SUBAPPLICATION InputOutputTesterButton_PI_OPC_UA (* PI Tester (OPC-UA): 8 Puls-Eingaenge (Zaehler+Frequenz+Bargraph) + 12 unveraenderte digitale Ausgaenge *)
  (* Standard: 61499-2; Description: Copyright (c) 2026 Meisterschulen am Ostbahnhof This program and the accompanying materials are made available under the terms of the Eclipse Public License 2.0 which is available at https://www.eclipse.org/legal/epl-2.0/ SPDX-License-Identifier: EPL-2.0 *)
  (* Version 1.0, 2026-08-30, Franz Höpfinger, Meisterschulen am Ostbahnhof, initial API and implementation and/or initial documentation *)
  PACKAGE Meins::InputOutputTester::Button_PI_OPC_UA;
  IMPORT Meins::InputOutputTester::Button_PI_OPC_UA::SubStrings::PI_I1_COUNT_WRITE;
  IMPORT Meins::InputOutputTester::Button_PI_OPC_UA::SubStrings::PI_I1_FREQ_WRITE;
  IMPORT Meins::InputOutputTester::Button_PI_OPC_UA::SubStrings::PI_I1_SWITCH_READ;
  IMPORT Meins::InputOutputTester::Button_PI_OPC_UA::SubStrings::PI_I1_SWITCH_WRITE;
  IMPORT Meins::InputOutputTester::Button_PI_OPC_UA::SubStrings::PI_I1_STATUS_WRITE;
  IMPORT Meins::InputOutputTester::Button_PI_OPC_UA::SubStrings::PI_I2_COUNT_WRITE;
  IMPORT Meins::InputOutputTester::Button_PI_OPC_UA::SubStrings::PI_I2_FREQ_WRITE;
  IMPORT Meins::InputOutputTester::Button_PI_OPC_UA::SubStrings::PI_I2_SWITCH_READ;
  IMPORT Meins::InputOutputTester::Button_PI_OPC_UA::SubStrings::PI_I2_SWITCH_WRITE;
  IMPORT Meins::InputOutputTester::Button_PI_OPC_UA::SubStrings::PI_I2_STATUS_WRITE;
  IMPORT Meins::InputOutputTester::Button_PI_OPC_UA::SubStrings::PI_I3_COUNT_WRITE;
  IMPORT Meins::InputOutputTester::Button_PI_OPC_UA::SubStrings::PI_I3_FREQ_WRITE;
  IMPORT Meins::InputOutputTester::Button_PI_OPC_UA::SubStrings::PI_I3_SWITCH_READ;
  IMPORT Meins::InputOutputTester::Button_PI_OPC_UA::SubStrings::PI_I3_SWITCH_WRITE;
  IMPORT Meins::InputOutputTester::Button_PI_OPC_UA::SubStrings::PI_I3_STATUS_WRITE;
  IMPORT Meins::InputOutputTester::Button_PI_OPC_UA::SubStrings::PI_I4_COUNT_WRITE;
  IMPORT Meins::InputOutputTester::Button_PI_OPC_UA::SubStrings::PI_I4_FREQ_WRITE;
  IMPORT Meins::InputOutputTester::Button_PI_OPC_UA::SubStrings::PI_I4_SWITCH_READ;
  IMPORT Meins::InputOutputTester::Button_PI_OPC_UA::SubStrings::PI_I4_SWITCH_WRITE;
  IMPORT Meins::InputOutputTester::Button_PI_OPC_UA::SubStrings::PI_I4_STATUS_WRITE;
  IMPORT Meins::InputOutputTester::Button_PI_OPC_UA::SubStrings::PI_I5_COUNT_WRITE;
  IMPORT Meins::InputOutputTester::Button_PI_OPC_UA::SubStrings::PI_I5_FREQ_WRITE;
  IMPORT Meins::InputOutputTester::Button_PI_OPC_UA::SubStrings::PI_I5_SWITCH_READ;
  IMPORT Meins::InputOutputTester::Button_PI_OPC_UA::SubStrings::PI_I5_SWITCH_WRITE;
  IMPORT Meins::InputOutputTester::Button_PI_OPC_UA::SubStrings::PI_I5_STATUS_WRITE;
  IMPORT Meins::InputOutputTester::Button_PI_OPC_UA::SubStrings::PI_I6_COUNT_WRITE;
  IMPORT Meins::InputOutputTester::Button_PI_OPC_UA::SubStrings::PI_I6_FREQ_WRITE;
  IMPORT Meins::InputOutputTester::Button_PI_OPC_UA::SubStrings::PI_I6_SWITCH_READ;
  IMPORT Meins::InputOutputTester::Button_PI_OPC_UA::SubStrings::PI_I6_SWITCH_WRITE;
  IMPORT Meins::InputOutputTester::Button_PI_OPC_UA::SubStrings::PI_I6_STATUS_WRITE;
  IMPORT Meins::InputOutputTester::Button_PI_OPC_UA::SubStrings::PI_I7_COUNT_WRITE;
  IMPORT Meins::InputOutputTester::Button_PI_OPC_UA::SubStrings::PI_I7_FREQ_WRITE;
  IMPORT Meins::InputOutputTester::Button_PI_OPC_UA::SubStrings::PI_I7_SWITCH_READ;
  IMPORT Meins::InputOutputTester::Button_PI_OPC_UA::SubStrings::PI_I7_SWITCH_WRITE;
  IMPORT Meins::InputOutputTester::Button_PI_OPC_UA::SubStrings::PI_I7_STATUS_WRITE;
  IMPORT Meins::InputOutputTester::Button_PI_OPC_UA::SubStrings::PI_I8_COUNT_WRITE;
  IMPORT Meins::InputOutputTester::Button_PI_OPC_UA::SubStrings::PI_I8_FREQ_WRITE;
  IMPORT Meins::InputOutputTester::Button_PI_OPC_UA::SubStrings::PI_I8_SWITCH_READ;
  IMPORT Meins::InputOutputTester::Button_PI_OPC_UA::SubStrings::PI_I8_SWITCH_WRITE;
  IMPORT Meins::InputOutputTester::Button_PI_OPC_UA::SubStrings::PI_I8_STATUS_WRITE;
  IMPORT Meins::InputOutputTester::Button_PI_OPC_UA::SubStrings::Q01_READ;
  IMPORT Meins::InputOutputTester::Button_PI_OPC_UA::SubStrings::Q01_WRITE;
  IMPORT Meins::InputOutputTester::Button_PI_OPC_UA::SubStrings::Q02_READ;
  IMPORT Meins::InputOutputTester::Button_PI_OPC_UA::SubStrings::Q02_WRITE;
  IMPORT Meins::InputOutputTester::Button_PI_OPC_UA::SubStrings::Q03_READ;
  IMPORT Meins::InputOutputTester::Button_PI_OPC_UA::SubStrings::Q03_WRITE;
  IMPORT Meins::InputOutputTester::Button_PI_OPC_UA::SubStrings::Q04_READ;
  IMPORT Meins::InputOutputTester::Button_PI_OPC_UA::SubStrings::Q04_WRITE;
  IMPORT Meins::InputOutputTester::Button_PI_OPC_UA::SubStrings::Q05_READ;
  IMPORT Meins::InputOutputTester::Button_PI_OPC_UA::SubStrings::Q05_WRITE;
  IMPORT Meins::InputOutputTester::Button_PI_OPC_UA::SubStrings::Q06_READ;
  IMPORT Meins::InputOutputTester::Button_PI_OPC_UA::SubStrings::Q06_WRITE;
  IMPORT Meins::InputOutputTester::Button_PI_OPC_UA::SubStrings::Q07_READ;
  IMPORT Meins::InputOutputTester::Button_PI_OPC_UA::SubStrings::Q07_WRITE;
  IMPORT Meins::InputOutputTester::Button_PI_OPC_UA::SubStrings::Q08_READ;
  IMPORT Meins::InputOutputTester::Button_PI_OPC_UA::SubStrings::Q08_WRITE;
  IMPORT Meins::InputOutputTester::Button_PI_OPC_UA::SubStrings::Q09_READ;
  IMPORT Meins::InputOutputTester::Button_PI_OPC_UA::SubStrings::Q09_WRITE;
  IMPORT Meins::InputOutputTester::Button_PI_OPC_UA::SubStrings::Q10_READ;
  IMPORT Meins::InputOutputTester::Button_PI_OPC_UA::SubStrings::Q10_WRITE;
  IMPORT Meins::InputOutputTester::Button_PI_OPC_UA::SubStrings::Q11_READ;
  IMPORT Meins::InputOutputTester::Button_PI_OPC_UA::SubStrings::Q11_WRITE;
  IMPORT Meins::InputOutputTester::Button_PI_OPC_UA::SubStrings::Q12_READ;
  IMPORT Meins::InputOutputTester::Button_PI_OPC_UA::SubStrings::Q12_WRITE;
  IMPORT Meins::InputOutputTester::Button_PI_OPC_UA::SubStrings::Tick_WRITE;
  IMPORT Uebungen::const::UT::PI::DefaultPool_PI_Numeric::NumberVariable_PI_FREQ_I01_N;
  IMPORT Uebungen::const::UT::PI::DefaultPool_PI_Numeric::NumberVariable_PI_FREQ_I02_N;
  IMPORT Uebungen::const::UT::PI::DefaultPool_PI_Numeric::NumberVariable_PI_FREQ_I03_N;
  IMPORT Uebungen::const::UT::PI::DefaultPool_PI_Numeric::NumberVariable_PI_FREQ_I04_N;
  IMPORT Uebungen::const::UT::PI::DefaultPool_PI_Numeric::NumberVariable_PI_FREQ_I05_N;
  IMPORT Uebungen::const::UT::PI::DefaultPool_PI_Numeric::NumberVariable_PI_FREQ_I06_N;
  IMPORT Uebungen::const::UT::PI::DefaultPool_PI_Numeric::NumberVariable_PI_FREQ_I07_N;
  IMPORT Uebungen::const::UT::PI::DefaultPool_PI_Numeric::NumberVariable_PI_FREQ_I08_N;
  IMPORT Uebungen::const::UT::PI::DefaultPool_PI::NumberVariable_PI_COUNT_I01;
  IMPORT Uebungen::const::UT::PI::DefaultPool_PI::NumberVariable_PI_COUNT_I02;
  IMPORT Uebungen::const::UT::PI::DefaultPool_PI::NumberVariable_PI_COUNT_I03;
  IMPORT Uebungen::const::UT::PI::DefaultPool_PI::NumberVariable_PI_COUNT_I04;
  IMPORT Uebungen::const::UT::PI::DefaultPool_PI::NumberVariable_PI_COUNT_I05;
  IMPORT Uebungen::const::UT::PI::DefaultPool_PI::NumberVariable_PI_COUNT_I06;
  IMPORT Uebungen::const::UT::PI::DefaultPool_PI::NumberVariable_PI_COUNT_I07;
  IMPORT Uebungen::const::UT::PI::DefaultPool_PI::NumberVariable_PI_COUNT_I08;
  IMPORT Uebungen::const::UT::PI::DefaultPool_PI::Button_PI_I01_SWITCH;
  IMPORT Uebungen::const::UT::PI::DefaultPool_PI::Button_PI_I01_STATUS;
  IMPORT Uebungen::const::UT::PI::DefaultPool_PI::Button_PI_I02_SWITCH;
  IMPORT Uebungen::const::UT::PI::DefaultPool_PI::Button_PI_I02_STATUS;
  IMPORT Uebungen::const::UT::PI::DefaultPool_PI::Button_PI_I03_SWITCH;
  IMPORT Uebungen::const::UT::PI::DefaultPool_PI::Button_PI_I03_STATUS;
  IMPORT Uebungen::const::UT::PI::DefaultPool_PI::Button_PI_I04_SWITCH;
  IMPORT Uebungen::const::UT::PI::DefaultPool_PI::Button_PI_I04_STATUS;
  IMPORT Uebungen::const::UT::PI::DefaultPool_PI::Button_PI_I05_SWITCH;
  IMPORT Uebungen::const::UT::PI::DefaultPool_PI::Button_PI_I05_STATUS;
  IMPORT Uebungen::const::UT::PI::DefaultPool_PI::Button_PI_I06_SWITCH;
  IMPORT Uebungen::const::UT::PI::DefaultPool_PI::Button_PI_I06_STATUS;
  IMPORT Uebungen::const::UT::PI::DefaultPool_PI::Button_PI_I07_SWITCH;
  IMPORT Uebungen::const::UT::PI::DefaultPool_PI::Button_PI_I07_STATUS;
  IMPORT Uebungen::const::UT::PI::DefaultPool_PI::Button_PI_I08_SWITCH;
  IMPORT Uebungen::const::UT::PI::DefaultPool_PI::Button_PI_I08_STATUS;
  IMPORT Uebungen::const::UT::PI::DefaultPool_PI::Button_Q01;
  IMPORT Uebungen::const::UT::PI::DefaultPool_PI::Button_Q02;
  IMPORT Uebungen::const::UT::PI::DefaultPool_PI::Button_Q03;
  IMPORT Uebungen::const::UT::PI::DefaultPool_PI::Button_Q04;
  IMPORT Uebungen::const::UT::PI::DefaultPool_PI::Button_Q05;
  IMPORT Uebungen::const::UT::PI::DefaultPool_PI::Button_Q06;
  IMPORT Uebungen::const::UT::PI::DefaultPool_PI::Button_Q07;
  IMPORT Uebungen::const::UT::PI::DefaultPool_PI::Button_Q08;
  IMPORT Uebungen::const::UT::PI::DefaultPool_PI::Button_Q09;
  IMPORT Uebungen::const::UT::PI::DefaultPool_PI::Button_Q10;
  IMPORT Uebungen::const::UT::PI::DefaultPool_PI::Button_Q11;
  IMPORT Uebungen::const::UT::PI::DefaultPool_PI::Button_Q12;
  IMPORT Uebungen::const::UT::PI::DefaultPool_PI::OutputNumber_Tick;
  IMPORT logiBUS::io::PI::logiBUS_PI::PulseInput_I1;
  IMPORT logiBUS::io::PI::logiBUS_PI::PulseInput_I2;
  IMPORT logiBUS::io::PI::logiBUS_PI::PulseInput_I3;
  IMPORT logiBUS::io::PI::logiBUS_PI::PulseInput_I4;
  IMPORT logiBUS::io::PI::logiBUS_PI::PulseInput_I5;
  IMPORT logiBUS::io::PI::logiBUS_PI::PulseInput_I6;
  IMPORT logiBUS::io::PI::logiBUS_PI::PulseInput_I7;
  IMPORT logiBUS::io::PI::logiBUS_PI::PulseInput_I8;
  IMPORT logiBUS::io::DQ::logiBUS_DO::Output_Q1;
  IMPORT logiBUS::io::DQ::logiBUS_DO::Output_Q10;
  IMPORT logiBUS::io::DQ::logiBUS_DO::Output_Q11;
  IMPORT logiBUS::io::DQ::logiBUS_DO::Output_Q12;
  IMPORT logiBUS::io::DQ::logiBUS_DO::Output_Q2;
  IMPORT logiBUS::io::DQ::logiBUS_DO::Output_Q3;
  IMPORT logiBUS::io::DQ::logiBUS_DO::Output_Q4;
  IMPORT logiBUS::io::DQ::logiBUS_DO::Output_Q5;
  IMPORT logiBUS::io::DQ::logiBUS_DO::Output_Q6;
  IMPORT logiBUS::io::DQ::logiBUS_DO::Output_Q7;
  IMPORT logiBUS::io::DQ::logiBUS_DO::Output_Q8;
  IMPORT logiBUS::io::DQ::logiBUS_DO::Output_Q9;
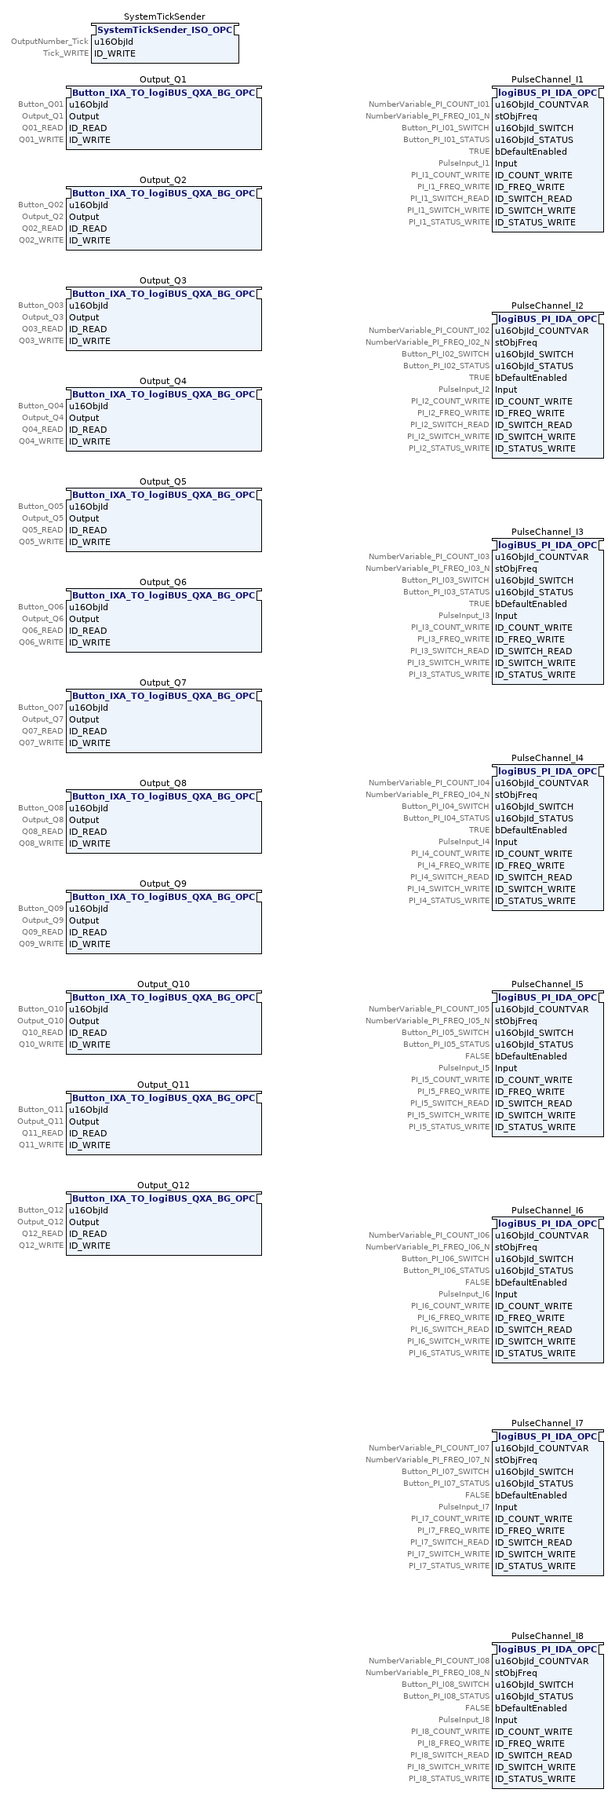
  SUBAPPS
    PulseChannel_I1 : MyLib::sys::logiBUS_PI_IDA_OPC(u16ObjId_COUNTVAR := NumberVariable_PI_COUNT_I01, stObjFreq := NumberVariable_PI_FREQ_I01_N, u16ObjId_SWITCH := Button_PI_I01_SWITCH, u16ObjId_STATUS := Button_PI_I01_STATUS, bDefaultEnabled := TRUE, Input := PulseInput_I1, ID_COUNT_WRITE := PI_I1_COUNT_WRITE, ID_FREQ_WRITE := PI_I1_FREQ_WRITE, ID_SWITCH_READ := PI_I1_SWITCH_READ, ID_SWITCH_WRITE := PI_I1_SWITCH_WRITE, ID_STATUS_WRITE := PI_I1_STATUS_WRITE);
    PulseChannel_I2 : MyLib::sys::logiBUS_PI_IDA_OPC(u16ObjId_COUNTVAR := NumberVariable_PI_COUNT_I02, stObjFreq := NumberVariable_PI_FREQ_I02_N, u16ObjId_SWITCH := Button_PI_I02_SWITCH, u16ObjId_STATUS := Button_PI_I02_STATUS, bDefaultEnabled := TRUE, Input := PulseInput_I2, ID_COUNT_WRITE := PI_I2_COUNT_WRITE, ID_FREQ_WRITE := PI_I2_FREQ_WRITE, ID_SWITCH_READ := PI_I2_SWITCH_READ, ID_SWITCH_WRITE := PI_I2_SWITCH_WRITE, ID_STATUS_WRITE := PI_I2_STATUS_WRITE);
    PulseChannel_I3 : MyLib::sys::logiBUS_PI_IDA_OPC(u16ObjId_COUNTVAR := NumberVariable_PI_COUNT_I03, stObjFreq := NumberVariable_PI_FREQ_I03_N, u16ObjId_SWITCH := Button_PI_I03_SWITCH, u16ObjId_STATUS := Button_PI_I03_STATUS, bDefaultEnabled := TRUE, Input := PulseInput_I3, ID_COUNT_WRITE := PI_I3_COUNT_WRITE, ID_FREQ_WRITE := PI_I3_FREQ_WRITE, ID_SWITCH_READ := PI_I3_SWITCH_READ, ID_SWITCH_WRITE := PI_I3_SWITCH_WRITE, ID_STATUS_WRITE := PI_I3_STATUS_WRITE);
    PulseChannel_I4 : MyLib::sys::logiBUS_PI_IDA_OPC(u16ObjId_COUNTVAR := NumberVariable_PI_COUNT_I04, stObjFreq := NumberVariable_PI_FREQ_I04_N, u16ObjId_SWITCH := Button_PI_I04_SWITCH, u16ObjId_STATUS := Button_PI_I04_STATUS, bDefaultEnabled := TRUE, Input := PulseInput_I4, ID_COUNT_WRITE := PI_I4_COUNT_WRITE, ID_FREQ_WRITE := PI_I4_FREQ_WRITE, ID_SWITCH_READ := PI_I4_SWITCH_READ, ID_SWITCH_WRITE := PI_I4_SWITCH_WRITE, ID_STATUS_WRITE := PI_I4_STATUS_WRITE);
    PulseChannel_I5 : MyLib::sys::logiBUS_PI_IDA_OPC(u16ObjId_COUNTVAR := NumberVariable_PI_COUNT_I05, stObjFreq := NumberVariable_PI_FREQ_I05_N, u16ObjId_SWITCH := Button_PI_I05_SWITCH, u16ObjId_STATUS := Button_PI_I05_STATUS, bDefaultEnabled := FALSE, Input := PulseInput_I5, ID_COUNT_WRITE := PI_I5_COUNT_WRITE, ID_FREQ_WRITE := PI_I5_FREQ_WRITE, ID_SWITCH_READ := PI_I5_SWITCH_READ, ID_SWITCH_WRITE := PI_I5_SWITCH_WRITE, ID_STATUS_WRITE := PI_I5_STATUS_WRITE);
    PulseChannel_I6 : MyLib::sys::logiBUS_PI_IDA_OPC(u16ObjId_COUNTVAR := NumberVariable_PI_COUNT_I06, stObjFreq := NumberVariable_PI_FREQ_I06_N, u16ObjId_SWITCH := Button_PI_I06_SWITCH, u16ObjId_STATUS := Button_PI_I06_STATUS, bDefaultEnabled := FALSE, Input := PulseInput_I6, ID_COUNT_WRITE := PI_I6_COUNT_WRITE, ID_FREQ_WRITE := PI_I6_FREQ_WRITE, ID_SWITCH_READ := PI_I6_SWITCH_READ, ID_SWITCH_WRITE := PI_I6_SWITCH_WRITE, ID_STATUS_WRITE := PI_I6_STATUS_WRITE);
    PulseChannel_I7 : MyLib::sys::logiBUS_PI_IDA_OPC(u16ObjId_COUNTVAR := NumberVariable_PI_COUNT_I07, stObjFreq := NumberVariable_PI_FREQ_I07_N, u16ObjId_SWITCH := Button_PI_I07_SWITCH, u16ObjId_STATUS := Button_PI_I07_STATUS, bDefaultEnabled := FALSE, Input := PulseInput_I7, ID_COUNT_WRITE := PI_I7_COUNT_WRITE, ID_FREQ_WRITE := PI_I7_FREQ_WRITE, ID_SWITCH_READ := PI_I7_SWITCH_READ, ID_SWITCH_WRITE := PI_I7_SWITCH_WRITE, ID_STATUS_WRITE := PI_I7_STATUS_WRITE);
    PulseChannel_I8 : MyLib::sys::logiBUS_PI_IDA_OPC(u16ObjId_COUNTVAR := NumberVariable_PI_COUNT_I08, stObjFreq := NumberVariable_PI_FREQ_I08_N, u16ObjId_SWITCH := Button_PI_I08_SWITCH, u16ObjId_STATUS := Button_PI_I08_STATUS, bDefaultEnabled := FALSE, Input := PulseInput_I8, ID_COUNT_WRITE := PI_I8_COUNT_WRITE, ID_FREQ_WRITE := PI_I8_FREQ_WRITE, ID_SWITCH_READ := PI_I8_SWITCH_READ, ID_SWITCH_WRITE := PI_I8_SWITCH_WRITE, ID_STATUS_WRITE := PI_I8_STATUS_WRITE);
    Output_Q1 : MyLib::sys::Button_IXA_TO_logiBUS_QXA_BG_OPC(u16ObjId := Button_Q01, Output := Output_Q1, ID_READ := Q01_READ, ID_WRITE := Q01_WRITE);
    Output_Q2 : MyLib::sys::Button_IXA_TO_logiBUS_QXA_BG_OPC(u16ObjId := Button_Q02, Output := Output_Q2, ID_READ := Q02_READ, ID_WRITE := Q02_WRITE);
    Output_Q3 : MyLib::sys::Button_IXA_TO_logiBUS_QXA_BG_OPC(u16ObjId := Button_Q03, Output := Output_Q3, ID_READ := Q03_READ, ID_WRITE := Q03_WRITE);
    Output_Q4 : MyLib::sys::Button_IXA_TO_logiBUS_QXA_BG_OPC(u16ObjId := Button_Q04, Output := Output_Q4, ID_READ := Q04_READ, ID_WRITE := Q04_WRITE);
    Output_Q5 : MyLib::sys::Button_IXA_TO_logiBUS_QXA_BG_OPC(u16ObjId := Button_Q05, Output := Output_Q5, ID_READ := Q05_READ, ID_WRITE := Q05_WRITE);
    Output_Q6 : MyLib::sys::Button_IXA_TO_logiBUS_QXA_BG_OPC(u16ObjId := Button_Q06, Output := Output_Q6, ID_READ := Q06_READ, ID_WRITE := Q06_WRITE);
    Output_Q7 : MyLib::sys::Button_IXA_TO_logiBUS_QXA_BG_OPC(u16ObjId := Button_Q07, Output := Output_Q7, ID_READ := Q07_READ, ID_WRITE := Q07_WRITE);
    Output_Q8 : MyLib::sys::Button_IXA_TO_logiBUS_QXA_BG_OPC(u16ObjId := Button_Q08, Output := Output_Q8, ID_READ := Q08_READ, ID_WRITE := Q08_WRITE);
    Output_Q9 : MyLib::sys::Button_IXA_TO_logiBUS_QXA_BG_OPC(u16ObjId := Button_Q09, Output := Output_Q9, ID_READ := Q09_READ, ID_WRITE := Q09_WRITE);
    Output_Q10 : MyLib::sys::Button_IXA_TO_logiBUS_QXA_BG_OPC(u16ObjId := Button_Q10, Output := Output_Q10, ID_READ := Q10_READ, ID_WRITE := Q10_WRITE);
    Output_Q11 : MyLib::sys::Button_IXA_TO_logiBUS_QXA_BG_OPC(u16ObjId := Button_Q11, Output := Output_Q11, ID_READ := Q11_READ, ID_WRITE := Q11_WRITE);
    Output_Q12 : MyLib::sys::Button_IXA_TO_logiBUS_QXA_BG_OPC(u16ObjId := Button_Q12, Output := Output_Q12, ID_READ := Q12_READ, ID_WRITE := Q12_WRITE);
    SystemTickSender : MyLib::sys::SystemTickSender_ISO_OPC(u16ObjId := OutputNumber_Tick, ID_WRITE := Tick_WRITE);
  END_SUBAPPS
END_SUBAPPLICATION
